PROGRAM MAIN
VAR
END_VAR

GVL.lamp := gvl.knop;

END_PROGRAM

(* stored: Version 1.1.0.1, ProductVersion 3.1.4024.12
   POU MAIN: Id {9eadf995-eec4-4666-bc62-ee440695cb18}, SpecialFunc None *)
